(* IEC 61131-3 sources: programs/VI-54/VI-54_20171205/VI-54_20171205/Stations/PLC_VI54/VI-54_171014/Class/ResetErrSafety, 1 file *)

(* ---- ResetErrSafety.st ---- *)
(*!
<Class
	Name               = "ResetErrSafety"
	Revision           = "0.0"
	RealtimeTask       = "false"
	CyclicTask         = "false"
	BackgroundTask     = "false"
	Sigmatek           = "false"
	OSInterface        = "false"
	HighPriority       = "false"
	Automatic          = "false"
	UpdateMode         = "Prescan"
	SharedCommandTable = "true"
	Objectsize         = "(450,180)">
	<Channels>
		<Server Name="Comm" Visualized="false" Initialize="false" WriteProtected="false" Retentive="false"/>
		<Client Name="iCheckErr" Required="true" Internal="false"/>
		<Client Name="oQuitCommErr" Required="true" Internal="false"/>
		<Client Name="Standard1" Required="true" Internal="true"/>
		<Client Name="TEST" Required="false" Internal="false"/>
	</Channels>
	<Network Name="ResetErrSafety">
		<!-- List of Components in this network -->
		<Components>
			<Object
				Name           = "Standard1"
				Class          = "Standard"
				Position       = "(360,180)"
				Visualized     = "false"
				BackgroundTime = "1000 ms">
				<Channels>
					<Server Name="ClassSvr"/>
				</Channels>
			</Object>
		</Components>
		<Comments>
		</Comments>
		<!-- List of Connections in this network -->
		<Connections>
			<Connection Source="this.Standard1" Destination="Standard1.ClassSvr"/>
		</Connections>
		<!-- Headerfiles -->
		<Options>
		</Options>
	</Network>
</Class>
*)
ResetErrSafety : CLASS
  //Servers:
	Comm 	: SvrChCmd_DINT;
  //Clients:
	iCheckErr 	: CltCh_DINT;
	oQuitCommErr 	: CltCh_DINT;
	Standard1 	: CltChCmd_Standard;
	TEST 	: CltCh_DINT;
  //Variables:
		ResetError 	: DINT;
  //Functions:

	FUNCTION VIRTUAL GLOBAL Comm::Write
		VAR_INPUT
			input (EAX) 	: DINT;
		END_VAR
		VAR_OUTPUT
			result (EAX) 	: DINT;
		END_VAR;
  //Tables:
	FUNCTION @STD
		VAR_OUTPUT
			ret_code	: CONFSTATES;
		END_VAR;
	FUNCTION GLOBAL TAB @CT_;
END_CLASS;

#pragma using Standard

FUNCTION VIRTUAL GLOBAL ResetErrSafety::Comm::Write
	VAR_INPUT
		input (EAX) 	: DINT;
	END_VAR
	VAR_OUTPUT
		result (EAX) 	: DINT;
	END_VAR

	Comm := input;

  // Check for error
  if TEST.Read() <> 0 then
    if Standard1.R_TRIG(CLK:= Comm) then
      oQuitCommErr := 1;
      oQuitCommErr.Write(input:= oQuitCommErr); // Write to output
    end_if;
  elsif Standard1.F_TRIG(CLK:= Comm) then
    oQuitCommErr := 0;
    oQuitCommErr.Write(input:= oQuitCommErr); // Write to output
  end_if;

END_FUNCTION
